// Mitsubishi GX Works2 project: 연습   PLC: Q03UDE

PROGRAM MAIN
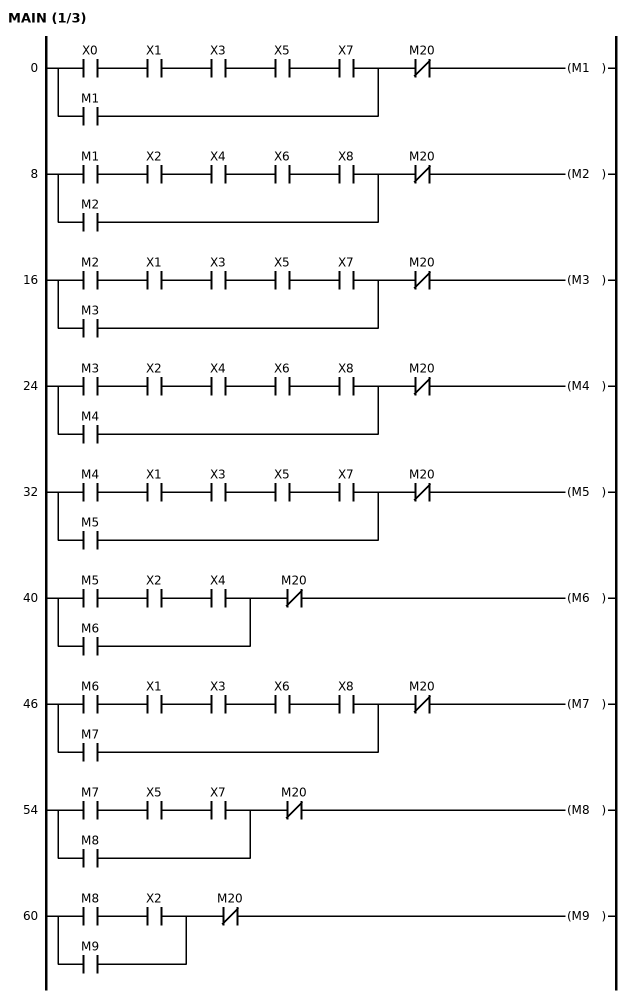
0     LD      X0
      AND     X1
      AND     X3
      AND     X5
      AND     X7
      OR      M1
      ANI     M20
      OUT     M1
8     LD      M1
      AND     X2
      AND     X4
      AND     X6
      AND     X8
      OR      M2
      ANI     M20
      OUT     M2
16    LD      M2
      AND     X1
      AND     X3
      AND     X5
      AND     X7
      OR      M3
      ANI     M20
      OUT     M3
24    LD      M3
      AND     X2
      AND     X4
      AND     X6
      AND     X8
      OR      M4
      ANI     M20
      OUT     M4
32    LD      M4
      AND     X1
      AND     X3
      AND     X5
      AND     X7
      OR      M5
      ANI     M20
      OUT     M5
40    LD      M5
      AND     X2
      AND     X4
      OR      M6
      ANI     M20
      OUT     M6
46    LD      M6
      AND     X1
      AND     X3
      AND     X6
      AND     X8
      OR      M7
      ANI     M20
      OUT     M7
54    LD      M7
      AND     X5
      AND     X7
      OR      M8
      ANI     M20
      OUT     M8
60    LD      M8
      AND     X2
      OR      M9
      ANI     M20
      OUT     M9
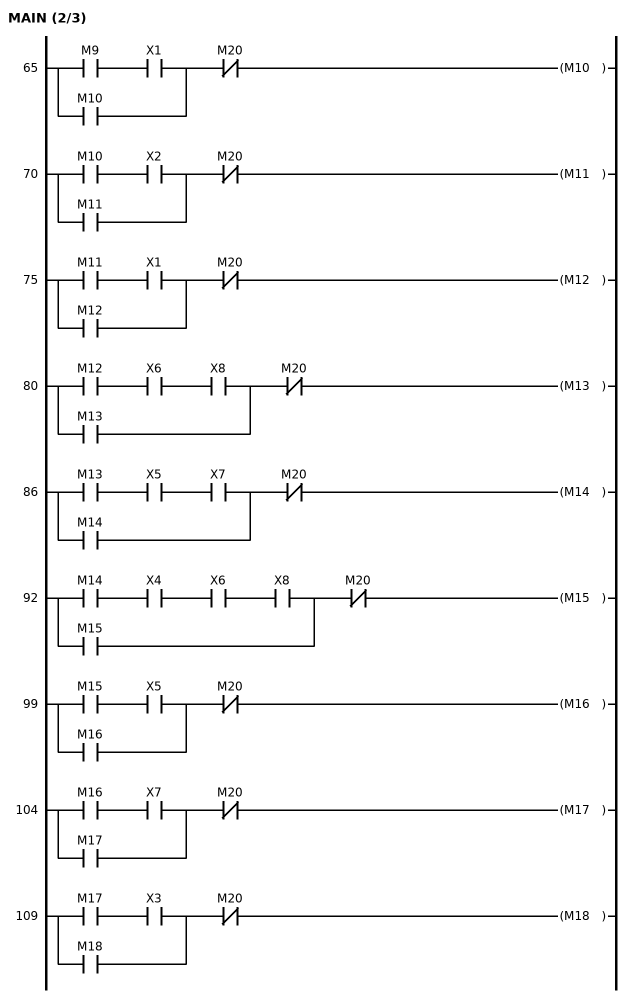
65    LD      M9
      AND     X1
      OR      M10
      ANI     M20
      OUT     M10
70    LD      M10
      AND     X2
      OR      M11
      ANI     M20
      OUT     M11
75    LD      M11
      AND     X1
      OR      M12
      ANI     M20
      OUT     M12
80    LD      M12
      AND     X6
      AND     X8
      OR      M13
      ANI     M20
      OUT     M13
86    LD      M13
      AND     X5
      AND     X7
      OR      M14
      ANI     M20
      OUT     M14
92    LD      M14
      AND     X4
      AND     X6
      AND     X8
      OR      M15
      ANI     M20
      OUT     M15
99    LD      M15
      AND     X5
      OR      M16
      ANI     M20
      OUT     M16
104   LD      M16
      AND     X7
      OR      M17
      ANI     M20
      OUT     M17
109   LD      M17
      AND     X3
      OR      M18
      ANI     M20
      OUT     M18
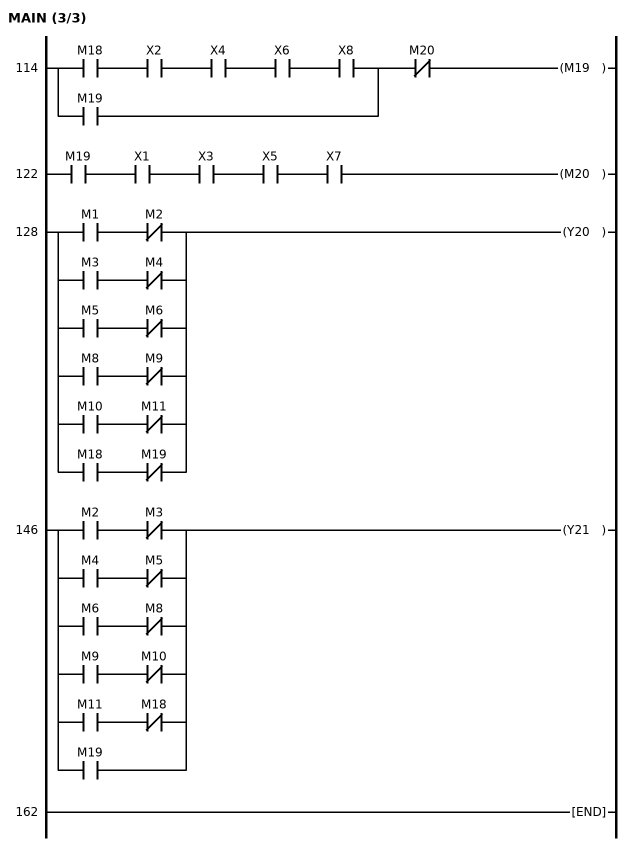
114   LD      M18
      AND     X2
      AND     X4
      AND     X6
      AND     X8
      OR      M19
      ANI     M20
      OUT     M19
122   LD      M19
      AND     X1
      AND     X3
      AND     X5
      AND     X7
      OUT     M20
128   LD      M1
      ANI     M2
      LD      M3
      ANI     M4
      ORB
      LD      M5
      ANI     M6
      ORB
      LD      M8
      ANI     M9
      ORB
      LD      M10
      ANI     M11
      ORB
      LD      M18
      ANI     M19
      ORB
      OUT     Y20
146   LD      M2
      ANI     M3
      LD      M4
      ANI     M5
      ORB
      LD      M6
      ANI     M8
      ORB
      LD      M9
      ANI     M10
      ORB
      LD      M11
      ANI     M18
      ORB
      OR      M19
      OUT     Y21
162   END
END_PROGRAM
